FUNCTION_BLOCK EVENTS
VAR_INPUT
	DATE_IN : DATE;
	ENA : BOOL;
END_VAR
VAR_OUTPUT
	Y : BOOL;
	NAME : STRING(30);
END_VAR
VAR
	i : INT;
	last_active : DATE;
	size :INT := 49;
	day_in: DINT;
	cyr: INT;
	lday: DINT;
	check : HOLIDAY_DATA;
	y_int : BOOL;
	name_int : STRING(30);
END_VAR
VAR_IN_OUT
	ELIST : ARRAY[0..49] OF HOLIDAY_DATA;
END_VAR

(*
version 1.0	18. jan. 2010
programmer 	hugo
tested by		tobias

event checks an array with a list of events and displays the event if today is one.

*)

(* for performance reasons only activate once a day *)
IF last_active <> date_in THEN
	last_active := DATE_IN;
	Y_int := FALSE;
	name_int := '';
	day_in := DAY_OF_DATE(DATE_IN);
	cyr := YEAR_OF_DATE(DATE_IN);

	(* search list for events *)
	FOR i := 0 TO size DO
		check := elist[i];
		lday := DAY_OF_DATE(SET_DATE(cyr,check.month, check.day));
		IF day_in >= lday AND day_in <= lday + check.use - 1 THEN
			y_int := TRUE;
			name_int := check.name;
			EXIT;
		END_IF;
	END_FOR;
END_IF;

IF ENA THEN
	Y := y_int;
	NAME := name_int;
ELSE
	Y := FALSE;
	NAME := '';
END_IF;

(* revision history
hm  18. jan. 2011	rev 1.0
	new module

*)

END_FUNCTION_BLOCK

(* stored: Version 1.1.0.1, ProductVersion 3.1.4022.7
   POU EVENTS: Id {87a884e6-6f76-48f3-bc8a-5ee41c4abb95}, SpecialFunc None *)
